FUNCTION_BLOCK FB_Module_ToolHolderDoor_Old IMPLEMENTS I_Module
VAR_INPUT
	bEnable					: BOOL;
END_VAR
VAR_OUTPUT
	bDoorUp				: BOOL;
END_VAR
VAR
	Components			: ARRAY [0..2] OF I_Component;
	
	fbPiston			: FB_Component_DualValve;
	fbDoorUp			: FB_Component_InductiveSensor;
	fbDoorDown			: FB_Component_ReedSwitch;
	idx					: INT;
END_VAR

IF bEnable THEN
	fbPiston(
		sName 		:= 'door piston',
		bEnable		:= TRUE,
		bOutputA	:= GVL.bCloseToolCarrierDoor,
		bOutputB	:= GVL.bOpenToolCarrierDoor);
	
	fbDoorUp(
		bRawSignal	:= GVL.bDoorToolHolderLock,
		tDebounce	:= T#0MS,
		tTimeout	:= T#0MS,
		sName		:= 'door up',
		bEnable		:= TRUE);
		
	fbDoorDown(
		bRawSignal	:= GVL.bDoorToolHolderDown,
		tDebounce	:= T#0MS,
		tTimeout	:= T#0MS,
		sName		:= 'door down',
		bEnable		:= TRUE);
		
	Components[0]	:= fbPiston;
	Components[1]	:= fbDoorUp;
	Components[2]	:= fbDoorDown;
	
	FOR idx := 0 TO 2 DO
    	Components[idx].M_Start();
	END_FOR;
	
	bDoorUp := fbDoorUp.bSensorActive;
END_IF

METHOD M_Down : BOOL
VAR_INPUT
END_VAR
IF bEnable THEN
	IF fbDoorDown.bSensorActive THEN
		fbPiston.M_Hold();
		M_Down := TRUE;
	ELSE
		fbPiston.M_Retract();
	END_IF
END_IF
END_METHOD

{warning 'add method implementation '}
METHOD M_Halt : BOOL
END_METHOD

{warning 'add method implementation '}
METHOD M_Start : BOOL
END_METHOD

{warning 'add method implementation '}
METHOD M_Stop : BOOL
END_METHOD

METHOD M_Up : BOOL
VAR_INPUT
END_VAR
IF bEnable THEN
	IF fbDoorUp.bSensorActive THEN
		fbPiston.M_Hold();
		M_Up := TRUE;
	ELSE
		fbPiston.M_Extend();
	END_IF
END_IF
END_METHOD

END_FUNCTION_BLOCK

(* stored: Version 1.1.0.1, ProductVersion 3.1.4024.15
   POU FB_Module_ToolHolderDoor_Old: Id {0d495e39-7cce-4183-99e5-9ac20d38389e}, SpecialFunc None
   Method M_Down: Id {b9e2c4a7-e1f6-4008-995a-5790ed9e33e3}
   Method M_Halt: Id {0b603238-625f-4883-b741-b13099fd28a6}
   Method M_Start: Id {027b75b5-29ad-4339-8c09-b924ca0fe761}
   Method M_Stop: Id {0c838a79-9df5-4a28-a13e-62b86fd1408b}
   Method M_Up: Id {390c175e-3aea-46f3-91f9-12aac5ce4f18} *)
